TYPE ST_Accelerometer :
STRUCT
	X: INT;
	Y: INT;
	Z: INT;
END_STRUCT
END_TYPE

(* stored: Version 1.1.0.1
   DUT ST_Accelerometer: Id {609788be-6cef-4bab-b82d-0de671123a2d} *)
